INTERFACE I_Command

METHOD Execute
END_METHOD

END_INTERFACE

(* stored: Version 1.1.0.1, ProductVersion 3.1.4019.2
   Itf I_Command: Id {b9552517-79a2-47e4-9ea4-093312b610dd}
   Method Execute: Id {8f5c6cfd-bac1-4bb2-8501-7a4064075c03} *)
